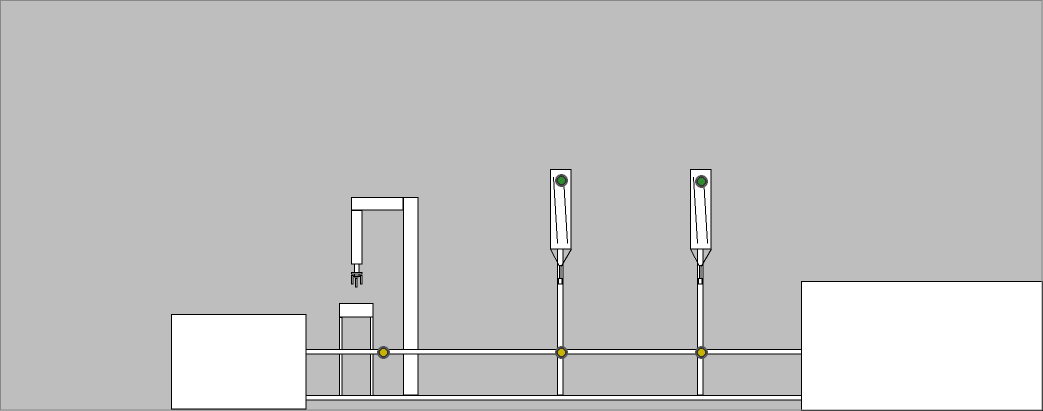
VISUALIZATION Visualization  // 1043x411
    Group (352,275 8x12), invisible if: NOT MAIN.MyMashine.MyRobot.RoboNagel.visible
        p3560616238: MAIN.MyMashine.MyRobot.i_HOZAxxe.i_i_AxxePosition
        p2738717112: MAIN.MyMashine.MyRobot.i_VTKAxxe.i_i_AxxePosition
        Ellipse (0,0 8x2)
        Rectangle (3,3 2x9)
    Rectangle (370,316 3x84)
    Rectangle (339,317 3x83)
    Rectangle (403,197 15x198)
    Rectangle (697,197 6x198)
    Rectangle (557,197 6x198)
    Rectangle (261,349 636x5)
    Rectangle (259,395 637x5)
    Ellipse (242,348 48x54)
    Group (293,327 8x12), invisible if: NOT MAIN.MyMashine.Holder[1].Nagel.visible
        p3560616238: MAIN.MyMashine.Holder[1].i_i_HolderPosition
        Ellipse (0,0 8x2)
        Rectangle (3,3 2x9)
    RoundedRectangle (290,339 13x10)
        p3560616238: MAIN.MyMashine.Holder[1].i_i_HolderPosition
    RoundedRectangle (290,339 13x10)
        p3560616238: MAIN.MyMashine.Holder[4].i_i_HolderPosition
    Group (293,327 8x12), invisible if: NOT MAIN.MyMashine.Holder[4].Nagel.visible
        p3560616238: MAIN.MyMashine.Holder[4].i_i_HolderPosition
        Ellipse (0,0 8x2)
        Rectangle (3,3 2x9)
    RoundedRectangle (290,339 13x10)
        p3560616238: MAIN.MyMashine.Holder[3].i_i_HolderPosition
    Group (293,327 8x12), invisible if: NOT MAIN.MyMashine.Holder[3].Nagel.visible
        p3560616238: MAIN.MyMashine.Holder[3].i_i_HolderPosition
        Ellipse (0,0 8x2)
        Rectangle (3,3 2x9)
    RoundedRectangle (290,339 13x10)
        p3560616238: MAIN.MyMashine.Holder[2].i_i_HolderPosition
    Group (293,327 8x12), invisible if: NOT MAIN.MyMashine.Holder[2].Nagel.visible
        p3560616238: MAIN.MyMashine.Holder[2].i_i_HolderPosition
        Ellipse (0,0 8x2)
        Rectangle (3,3 2x9)
    Rectangle (351,197 52x13)
    Group (351,210 11x74)
        p3560616238: MAIN.MyMashine.MyRobot.i_HOZAxxe.i_i_AxxePosition
        Rectangle (9,65 2x9)
            p3560616238: MAIN.MyMashine.MyRobot.i_GRFRightAxxe.i_i_AxxePosition
            p2738717112: MAIN.MyMashine.MyRobot.i_VTKAxxe.i_i_AxxePosition
        Rectangle (0,65 2x9)
            p3560616238: MAIN.MyMashine.MyRobot.i_GRFLeftAxxe.i_i_AxxePosition
            p2738717112: MAIN.MyMashine.MyRobot.i_VTKAxxe.i_i_AxxePosition
        Rectangle (3,1 5x65)
            p2738717112: MAIN.MyMashine.MyRobot.i_VTKAxxe.i_i_AxxePosition
        Rectangle (0,62 11x2)
            p2738717112: MAIN.MyMashine.MyRobot.i_VTKAxxe.i_i_AxxePosition
        Rectangle (0,0 11x54)
    Group (550,169 21x115)
        p2738717112: MAIN.MyMashine.l_Schraubendreher1.i_VTKAxxe.i_i_AxxePosition
        Rectangle (0,0 21x80)
        Line (21,80) (11,97)
        Line (0,80) (9,97)
        RoundedRectangle (9,96 2x14)
        Rectangle (8,109 4x6)
        Line (13,8) (17,74)
        Line (3,8) (7,74)
        Lamp1 (4,4 15x15), variable: MAIN.MyMashine.l_Schraubendreher1.l_b_Power, style: Lamp-Lamp1-Green
    Group (690,169 21x115)
        p2738717112: MAIN.MyMashine.l_Schraubendreher2.i_VTKAxxe.i_i_AxxePosition
        Rectangle (0,0 21x80)
        Line (21,80) (11,97)
        Line (0,80) (9,97)
        RoundedRectangle (9,96 2x14)
        Rectangle (8,109 4x6)
        Line (13,8) (17,74)
        Line (3,8) (7,74)
        Lamp1 (4,5 15x15), variable: MAIN.MyMashine.l_Schraubendreher2.l_b_Power, style: Lamp-Lamp1-Green
    Lamp1 (554,345 15x15), variable: MAIN.MyMashine.Sensore2.i_b_SensoreActive, style: Lamp-Lamp1-Yellow
    Lamp1 (694,345 15x15), variable: MAIN.MyMashine.Sensore3.i_b_SensoreActive, style: Lamp-Lamp1-Yellow
    Rectangle (339,303 34x14)
    RoundedRectangle (290,338 13x10)
        p3560616238: MAIN.MyMashine.Holder[11].i_i_HolderPosition
    Group (293,326 8x12), invisible if: NOT MAIN.MyMashine.Holder[2].Nagel.visible
        p3560616238: MAIN.MyMashine.Holder[11].i_i_HolderPosition
        Ellipse (0,0 8x2)
        Rectangle (3,3 2x9)
    RoundedRectangle (290,339 13x10)
        p3560616238: MAIN.MyMashine.Holder[9].i_i_HolderPosition
    Group (293,327 8x12), invisible if: NOT MAIN.MyMashine.Holder[2].Nagel.visible
        p3560616238: MAIN.MyMashine.Holder[9].i_i_HolderPosition
        Ellipse (0,0 8x2)
        Rectangle (3,3 2x9)
    RoundedRectangle (291,339 13x10)
        p3560616238: MAIN.MyMashine.Holder[8].i_i_HolderPosition
    Group (294,325 8x12), invisible if: NOT MAIN.MyMashine.Holder[8].Nagel.visible
        p3560616238: MAIN.MyMashine.Holder[8].i_i_HolderPosition
        Ellipse (0,0 8x2)
        Rectangle (3,3 2x9)
    RoundedRectangle (290,339 13x10)
        p3560616238: MAIN.MyMashine.Holder[7].i_i_HolderPosition
    Group (293,327 8x12), invisible if: NOT MAIN.MyMashine.Holder[7].Nagel.visible
        p3560616238: MAIN.MyMashine.Holder[7].i_i_HolderPosition
        Ellipse (0,0 8x2)
        Rectangle (3,3 2x9)
    RoundedRectangle (291,339 13x10)
        p3560616238: MAIN.MyMashine.Holder[6].i_i_HolderPosition
    Group (294,327 8x12), invisible if: NOT MAIN.MyMashine.Holder[6].Nagel.visible
        p3560616238: MAIN.MyMashine.Holder[6].i_i_HolderPosition
        Ellipse (0,0 8x2)
        Rectangle (3,3 2x9)
    RoundedRectangle (290,339 13x10)
        p3560616238: MAIN.MyMashine.Holder[5].i_i_HolderPosition
    Group (293,326 8x12), invisible if: NOT MAIN.MyMashine.Holder[5].Nagel.visible
        p3560616238: MAIN.MyMashine.Holder[5].i_i_HolderPosition
        Ellipse (0,0 8x2)
        Rectangle (3,3 2x9)
    Lamp1 (376,345 15x15), variable: MAIN.MyMashine.Sensore1.i_b_SensoreActive, style: Lamp-Lamp1-Yellow
    Rectangle (801,281 242x130)
    Rectangle (171,314 135x95)
END_VISUALIZATION

(* stored: Version 1.1.0.1, ProductVersion 3.1.4024.3
   Visu Visualization: Id {e86d4129-978c-4f4f-b5db-62e336a35b6a} *)
